TYPE ST_MotionParameters :
STRUCT
	fSpeed		:	LREAL,
	tExpoTime	:	TIME
END_STRUCT
END_TYPE

(* stored: Version 1.1.0.1, ProductVersion 3.1.4022.18
   DUT ST_MotionParameters: Id {5b9a74fd-306c-4f18-884a-e0d91b09c5da} *)
